(* Logix 5000 project; controller TEC_81 vendor 1 type 14 code 148 rev 36.11; software revision 36.00; part 4 of 5 *)
(* tags used below, declared in another part *)
   AbrirInterlock_conveyor_Safety : BOOL;   // Mapped green button for interlock 2 opening
   AbrirInterlock_Principal_Safety : BOOL;   // Mapped green button for interlock 1 opening
   EStops_OK : BOOL;   // E-Stop Close Loop Indicator
   Interlocks_Ok : BOOL;   // Interlocks Close Loop Indicator
   LigthCurtain_ok : BOOL;   // Light Curtains Close Loop Indicator
   MC_1_EStop : DCI_STOP;   // Status of E-Stop 1
   MC_1_EStop_Status : BOOL;   // General status of inputs
   MC_1_Interlock : DCI_STOP;   // Status of Interlock 1
   MC_1_Interlock_Status : BOOL;   // General status of inputs
   MC_1_LigthCurtain : DCI_STOP;   // Status of Light Curtain 1
   MC_1_LigthCurtain_Status : BOOL;   // General status of inputs
   MC_2_EStop : DCI_STOP;   // Status of E-Stop 2
   MC_2_EStop_Status : BOOL;   // General status of inputs
   MC_2_Interlock : DCI_STOP;   // Status of Interlock 2
   MC_2_Interlock_Status : BOOL;   // General status of inputs
   MC_2_LightCurtain_Status : BOOL;   // General status of inputs
   MC_2_LigthCurtain : DCI_STOP;   // Status of Light Curtain 2
   MC_3_EStop : DCI_STOP;   // Status of E-Stop 3
   MC_3_EStop_Status : BOOL;   // General status of inputs
   MC_4_EStop : DCI_STOP;   // Status of E-Stop 4
   MC_4_EStop_Status : BOOL;   // General status of inputs
   MC_5_EStop : DCI_STOP;   // Status of E-Stop 5
   MC_5_EStop_Status : BOOL;   // General status of inputs
   ok : BOOL;
   Ons : INT;
   Operation_Mode : BOOL;   // Operation Mode for HMI (1) Manual (0) Automatico
   Paro_Emergencia_Almacen_1 : BOOL;   // Stopping signal of Torc Off Almacen 1
   Paro_Emergencia_Almacen_2 : BOOL;   // Stopping signal of Torc Off Almacen 2
   Reset_Almacen_1_Sfty : BOOL;
   Reset_Almacen_2_Sfty : BOOL;
   Reset_Principal_Sfty : BOOL;
   Reset_Salida_1_Sfty : BOOL;
   Safety_FromTEC81 : Safety;
   SafetyReset_almacen_1 : BOOL;   // Reset status Almacen 1
   SafetyReset_almacen_2 : BOOL;   // Reset status Almacen 2
   SafetyReset_Principal : BOOL;   // Reset status salida principal
   SafetyReset_Salida_1 : BOOL;   // Reset status Salida 1
   Storage_2 : BOOL;
   Storage_3 : BOOL;
   Storage_4 : BOOL;
   Storage_5 : BOOL;
   test_com : BOOL;   // bit e comunicacion
   TEst_Leaa_Sfty : DINT;
   TOF_STO_KinetixStorage2 : TIMER;
   TT : BOOL;

PROGRAM SafetyProgram   (* main routine MainRoutine, safety *)
VAR
   dummy : BOOL;
   Lasers_OK : BOOL;   // Laser Scanner Close Loop Indicator
   LS_1 : DCI_STOP := (InputStatus := 1, RestartType := 1, ColdStartType := 1, SafetyFunction := 1, DiscrepancyTime := 200);   // Status of Laser Scanner 1
   LS_1_Status : BOOL := 1;   // General status of inputs
   LS_2 : DCI_STOP := (ChannelA := 1, ChannelB := 1, InputStatus := 1, RestartType := 1, ColdStartType := 1, SafetyFunction := 1, DiscrepancyTime := 200, O1 := 1);   // Status of Laser Scanner 2
   LS_2_Status : BOOL := 1;   // General status of inputs
   Mat_1 : DCI_STOP := (InputStatus := 1, RestartType := 1, ColdStartType := 1, SafetyFunction := 4, DiscrepancyTime := 200);   // Status of Safety Mat 1
   Mat_1_Status : BOOL := 1;   // General status of inputs
   ONS_Laser_1 : BOOL;   // One time execution for reset
   ONS_Laser_2 : BOOL;   // One time execution for reset
   ONS_Mat_1 : BOOL;   // One time execution for reset
   Output_Enable_Laser_1 : BOOL;   // General status of Laser 1
   Output_Enable_Laser_2 : BOOL;   // General status of Laser 2
   Output_Enable_Mat_1 : BOOL;   // General status of Mat 1
   Safety_Close_Loop_ok : BOOL := 1;   // General Safety Indicator
   Safety_Latch_Timer : TIMER := (PRE := 500);
   Safety_Mat_ok : BOOL;   // Safety Mat Close Loop Indicator
   Safety_Reset_General : BOOL;   // Unified General Reset
   test_1 : BOOL;
   test_21 : BOOL;
   TOF_STO_KinetixStorage1 : TIMER := (PRE := 10000, EN := 1, DN := 1);
END_VAR

ROUTINE Almacenes   (* ladder *)
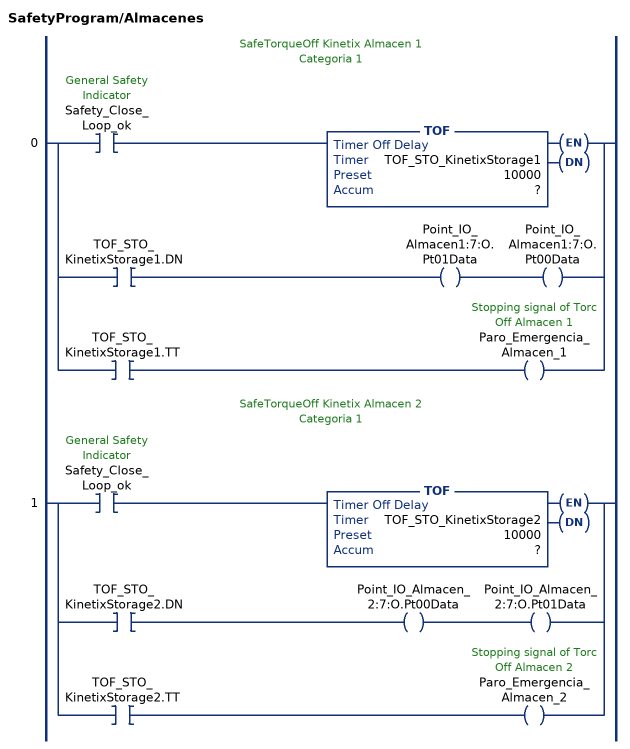
   // SafeTorqueOff Kinetix Almacen 1
   // Categoria 1
   0: [XIC(Safety_Close_Loop_ok) TOF(TOF_STO_KinetixStorage1,?,?) ,XIC(TOF_STO_KinetixStorage1.DN) OTE(Point_IO_Almacen1:7:O.Pt01Data) OTE(Point_IO_Almacen1:7:O.Pt00Data) ,XIC(TOF_STO_KinetixStorage1.TT) OTE(Paro_Emergencia_Almacen_1) ];
   // SafeTorqueOff Kinetix Almacen 2
   // Categoria 1
   1: [XIC(Safety_Close_Loop_ok) TOF(TOF_STO_KinetixStorage2,?,?) ,XIC(TOF_STO_KinetixStorage2.DN) OTE(Point_IO_Almacen_2:7:O.Pt00Data) OTE(Point_IO_Almacen_2:7:O.Pt01Data) ,XIC(TOF_STO_KinetixStorage2.TT) OTE(Paro_Emergencia_Almacen_2) ];
END_ROUTINE

ROUTINE Conveyors   (* ladder *)
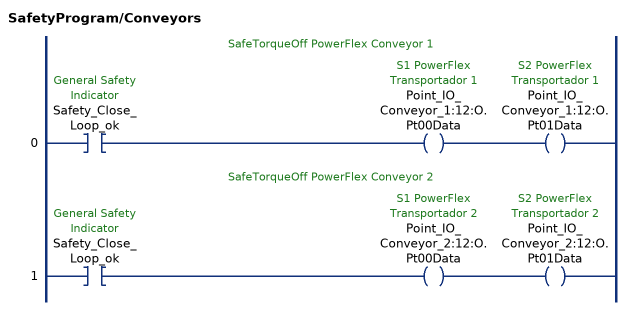
   // SafeTorqueOff PowerFlex Conveyor 1
   0: XIC(Safety_Close_Loop_ok)OTE(Point_IO_Conveyor_1:12:O.Pt00Data)OTE(Point_IO_Conveyor_1:12:O.Pt01Data);
   // SafeTorqueOff PowerFlex Conveyor 2
   1: XIC(Safety_Close_Loop_ok)OTE(Point_IO_Conveyor_2:12:O.Pt00Data)OTE(Point_IO_Conveyor_2:12:O.Pt01Data);
END_ROUTINE

ROUTINE Estops   (* ladder *)
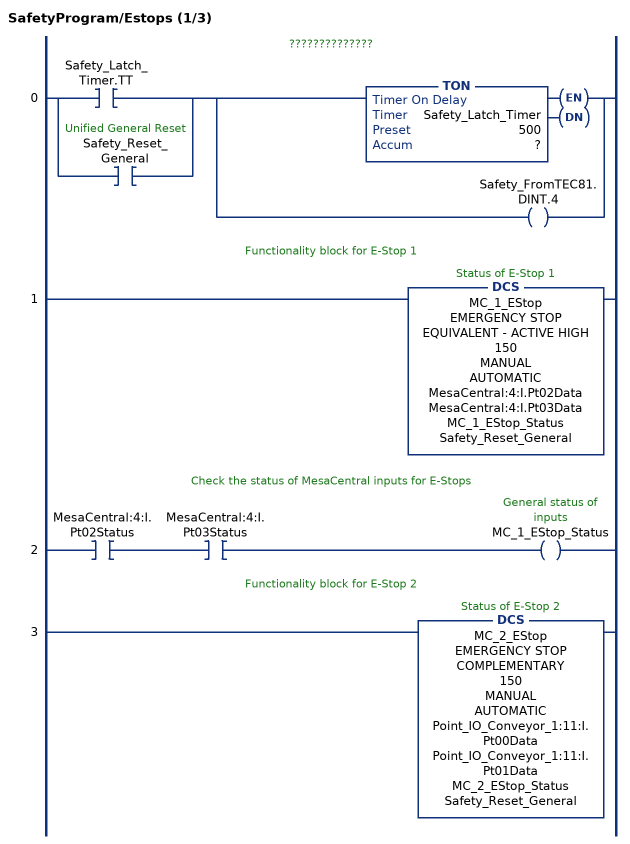
   // ??????????????
   0: [XIC(Safety_Latch_Timer.TT) ,XIC(Safety_Reset_General) ][TON(Safety_Latch_Timer,?,?) ,OTE(Safety_FromTEC81.DINT.4) ];
   // Functionality block for E-Stop 1
   1: DCS(MC_1_EStop,EMERGENCY STOP,EQUIVALENT - ACTIVE HIGH,150,MANUAL,AUTOMATIC,MesaCentral:4:I.Pt02Data,MesaCentral:4:I.Pt03Data,MC_1_EStop_Status,Safety_Reset_General);
   // Check the status of MesaCentral inputs for E-Stops
   2: XIC(MesaCentral:4:I.Pt02Status)XIC(MesaCentral:4:I.Pt03Status)OTE(MC_1_EStop_Status);
   // Functionality block for E-Stop 2
   3: DCS(MC_2_EStop,EMERGENCY STOP,COMPLEMENTARY,150,MANUAL,AUTOMATIC,Point_IO_Conveyor_1:11:I.Pt00Data,Point_IO_Conveyor_1:11:I.Pt01Data,MC_2_EStop_Status,Safety_Reset_General);
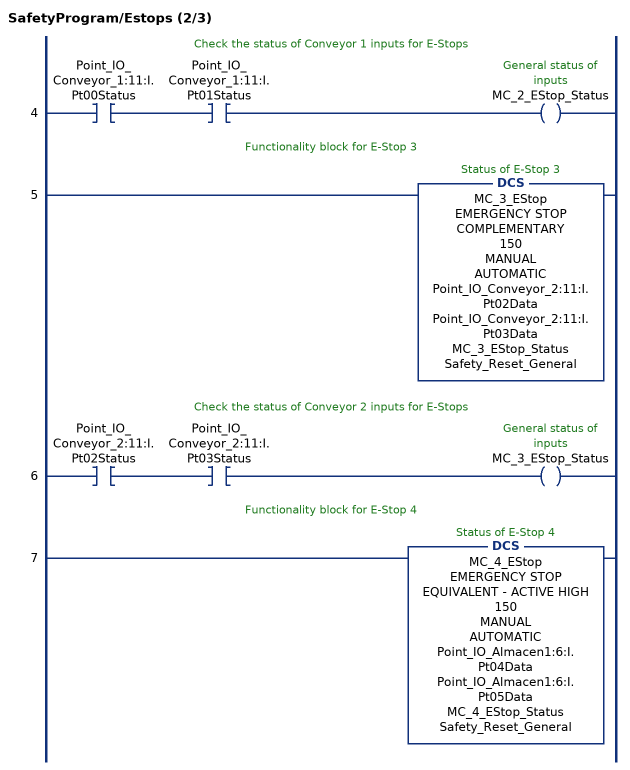
   // Check the status of Conveyor 1 inputs for E-Stops
   4: XIC(Point_IO_Conveyor_1:11:I.Pt00Status)XIC(Point_IO_Conveyor_1:11:I.Pt01Status)OTE(MC_2_EStop_Status);
   // Functionality block for E-Stop 3
   5: DCS(MC_3_EStop,EMERGENCY STOP,COMPLEMENTARY,150,MANUAL,AUTOMATIC,Point_IO_Conveyor_2:11:I.Pt02Data,Point_IO_Conveyor_2:11:I.Pt03Data,MC_3_EStop_Status,Safety_Reset_General);
   // Check the status of Conveyor 2 inputs for E-Stops
   6: XIC(Point_IO_Conveyor_2:11:I.Pt02Status)XIC(Point_IO_Conveyor_2:11:I.Pt03Status)OTE(MC_3_EStop_Status);
   // Functionality block for E-Stop 4
   7: DCS(MC_4_EStop,EMERGENCY STOP,EQUIVALENT - ACTIVE HIGH,150,MANUAL,AUTOMATIC,Point_IO_Almacen1:6:I.Pt04Data,Point_IO_Almacen1:6:I.Pt05Data,MC_4_EStop_Status,Safety_Reset_General);
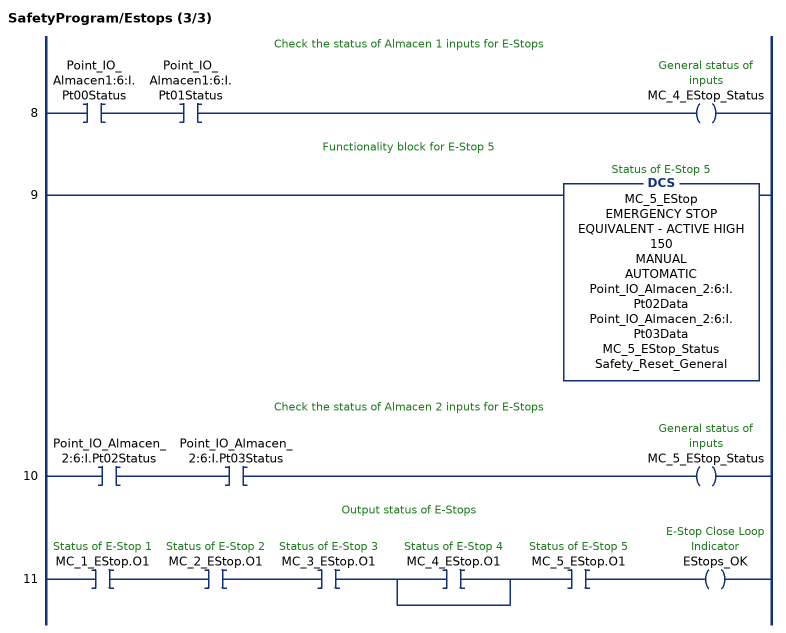
   // Check the status of Almacen 1 inputs for E-Stops
   8: XIC(Point_IO_Almacen1:6:I.Pt00Status)XIC(Point_IO_Almacen1:6:I.Pt01Status)OTE(MC_4_EStop_Status);
   // Functionality block for E-Stop 5
   9: DCS(MC_5_EStop,EMERGENCY STOP,EQUIVALENT - ACTIVE HIGH,150,MANUAL,AUTOMATIC,Point_IO_Almacen_2:6:I.Pt02Data,Point_IO_Almacen_2:6:I.Pt03Data,MC_5_EStop_Status,Safety_Reset_General);
   // Check the status of Almacen 2 inputs for E-Stops
   10: XIC(Point_IO_Almacen_2:6:I.Pt02Status)XIC(Point_IO_Almacen_2:6:I.Pt03Status)OTE(MC_5_EStop_Status);
   // Output status of E-Stops
   11: XIC(MC_1_EStop.O1)XIC(MC_2_EStop.O1)XIC(MC_3_EStop.O1)[XIC(MC_4_EStop.O1) ,]XIC(MC_5_EStop.O1)OTE(EStops_OK);
END_ROUTINE

ROUTINE External_COMM   (* ladder *)
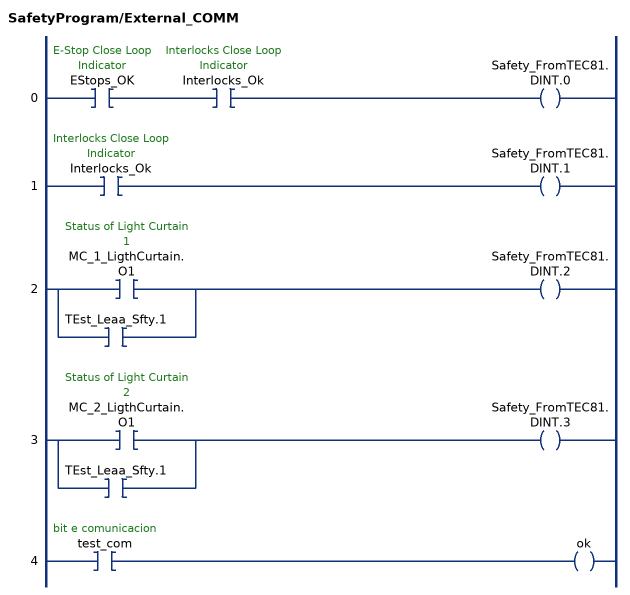
   0: XIC(EStops_OK)XIC(Interlocks_Ok)OTE(Safety_FromTEC81.DINT.0);
   1: XIC(Interlocks_Ok)OTE(Safety_FromTEC81.DINT.1);
   2: [XIC(MC_1_LigthCurtain.O1) ,XIC(TEst_Leaa_Sfty.1) ]OTE(Safety_FromTEC81.DINT.2);
   3: [XIC(MC_2_LigthCurtain.O1) ,XIC(TEst_Leaa_Sfty.1) ]OTE(Safety_FromTEC81.DINT.3);
   4: XIC(test_com)OTE(ok);
END_ROUTINE

ROUTINE Fanuc_Delta   (* ladder *)
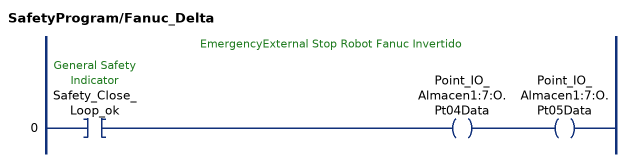
   // EmergencyExternal Stop Robot Fanuc Invertido
   0: XIC(Safety_Close_Loop_ok)OTE(Point_IO_Almacen1:7:O.Pt04Data)OTE(Point_IO_Almacen1:7:O.Pt05Data);
END_ROUTINE

ROUTINE Fanuc_Invertido   (* ladder *)
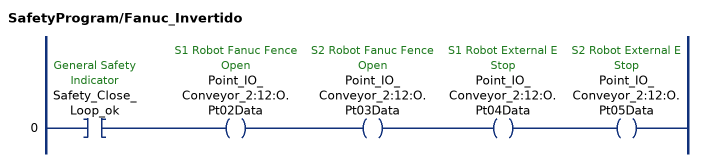
   0: XIC(Safety_Close_Loop_ok)OTE(Point_IO_Conveyor_2:12:O.Pt02Data)OTE(Point_IO_Conveyor_2:12:O.Pt03Data)OTE(Point_IO_Conveyor_2:12:O.Pt04Data)OTE(Point_IO_Conveyor_2:12:O.Pt05Data);
END_ROUTINE

ROUTINE Interlocks   (* ladder *)
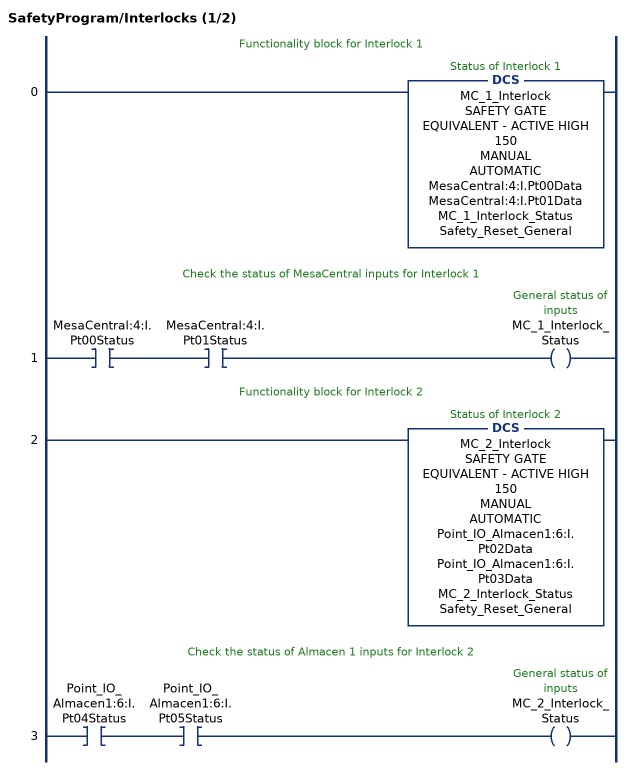
   // Functionality block for Interlock 1
   0: DCS(MC_1_Interlock,SAFETY GATE,EQUIVALENT - ACTIVE HIGH,150,MANUAL,AUTOMATIC,MesaCentral:4:I.Pt00Data,MesaCentral:4:I.Pt01Data,MC_1_Interlock_Status,Safety_Reset_General);
   // Check the status of MesaCentral inputs for Interlock 1
   1: XIC(MesaCentral:4:I.Pt00Status)XIC(MesaCentral:4:I.Pt01Status)OTE(MC_1_Interlock_Status);
   // Functionality block for Interlock 2
   2: DCS(MC_2_Interlock,SAFETY GATE,EQUIVALENT - ACTIVE HIGH,150,MANUAL,AUTOMATIC,Point_IO_Almacen1:6:I.Pt02Data,Point_IO_Almacen1:6:I.Pt03Data,MC_2_Interlock_Status,Safety_Reset_General);
   // Check the status of Almacen 1 inputs for Interlock 2
   3: XIC(Point_IO_Almacen1:6:I.Pt04Status)XIC(Point_IO_Almacen1:6:I.Pt05Status)OTE(MC_2_Interlock_Status);
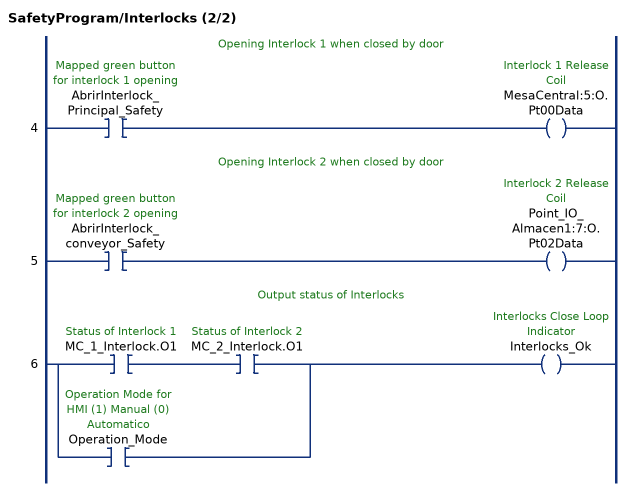
   // Opening Interlock 1 when closed by door
   4: XIC(AbrirInterlock_Principal_Safety)OTE(MesaCentral:5:O.Pt00Data);
   // Opening Interlock 2 when closed by door
   5: XIC(AbrirInterlock_conveyor_Safety)OTE(Point_IO_Almacen1:7:O.Pt02Data);
   // Output status of Interlocks
   6: [XIC(MC_1_Interlock.O1) XIC(MC_2_Interlock.O1) ,XIC(Operation_Mode) ]OTE(Interlocks_Ok);
END_ROUTINE

ROUTINE Laser_Scanner   (* ladder *)
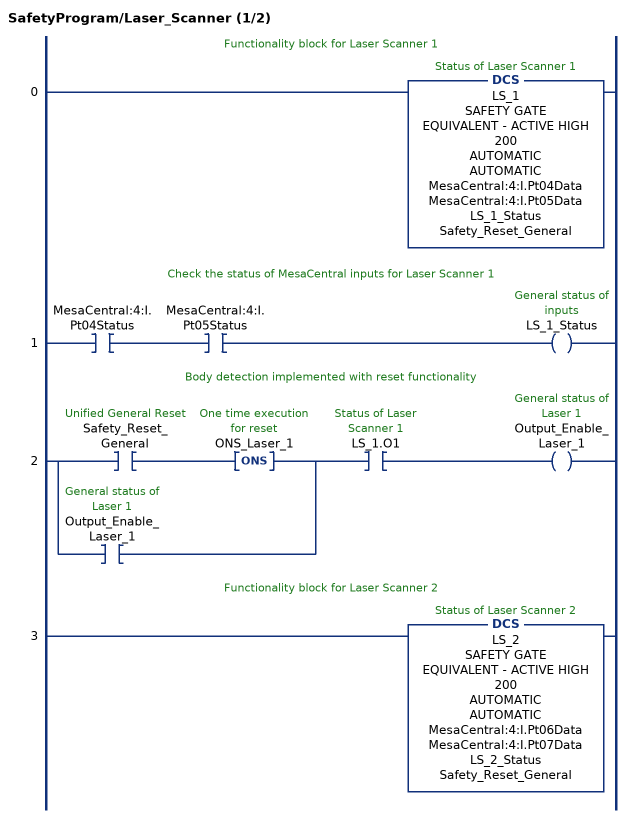
   // Functionality block for Laser Scanner 1
   0: DCS(LS_1,SAFETY GATE,EQUIVALENT - ACTIVE HIGH,200,AUTOMATIC,AUTOMATIC,MesaCentral:4:I.Pt04Data,MesaCentral:4:I.Pt05Data,LS_1_Status,Safety_Reset_General);
   // Check the status of MesaCentral inputs for Laser Scanner 1
   1: XIC(MesaCentral:4:I.Pt04Status)XIC(MesaCentral:4:I.Pt05Status)OTE(LS_1_Status);
   // Body detection implemented with reset functionality
   2: [XIC(Safety_Reset_General) ONS(ONS_Laser_1) ,XIC(Output_Enable_Laser_1) ]XIC(LS_1.O1)OTE(Output_Enable_Laser_1);
   // Functionality block for Laser Scanner 2
   3: DCS(LS_2,SAFETY GATE,EQUIVALENT - ACTIVE HIGH,200,AUTOMATIC,AUTOMATIC,MesaCentral:4:I.Pt06Data,MesaCentral:4:I.Pt07Data,LS_2_Status,Safety_Reset_General);
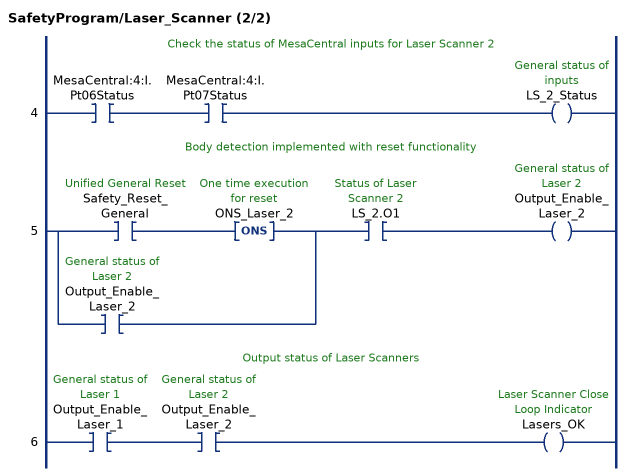
   // Check the status of MesaCentral inputs for Laser Scanner 2
   4: XIC(MesaCentral:4:I.Pt06Status)XIC(MesaCentral:4:I.Pt07Status)OTE(LS_2_Status);
   // Body detection implemented with reset functionality
   5: [XIC(Safety_Reset_General) ONS(ONS_Laser_2) ,XIC(Output_Enable_Laser_2) ]XIC(LS_2.O1)OTE(Output_Enable_Laser_2);
   // Output status of Laser Scanners
   6: XIC(Output_Enable_Laser_1)XIC(Output_Enable_Laser_2)OTE(Lasers_OK);
END_ROUTINE

ROUTINE LigthCurrtains   (* ladder *)
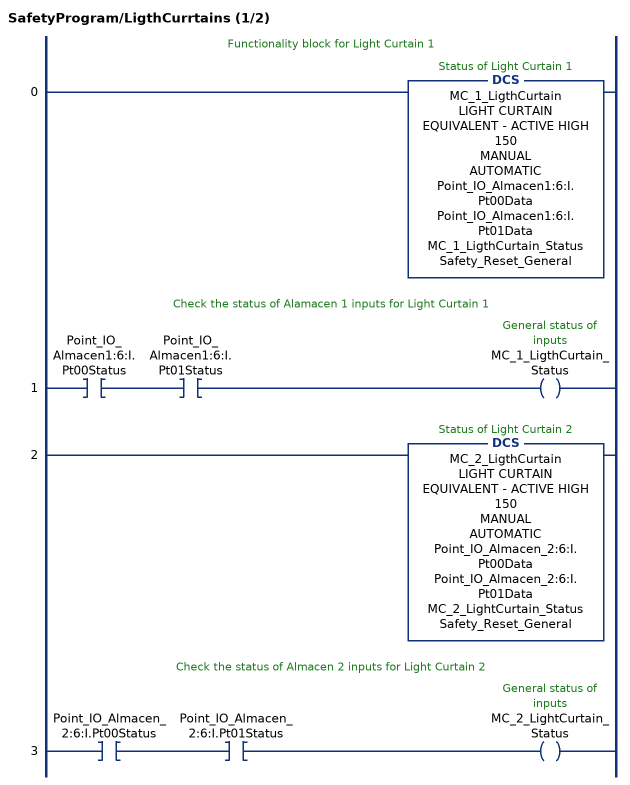
   // Functionality block for Light Curtain 1
   0: DCS(MC_1_LigthCurtain,LIGHT CURTAIN,EQUIVALENT - ACTIVE HIGH,150,MANUAL,AUTOMATIC,Point_IO_Almacen1:6:I.Pt00Data,Point_IO_Almacen1:6:I.Pt01Data,MC_1_LigthCurtain_Status,Safety_Reset_General);
   // Check the status of Alamacen 1 inputs for Light Curtain 1
   1: XIC(Point_IO_Almacen1:6:I.Pt00Status)XIC(Point_IO_Almacen1:6:I.Pt01Status)OTE(MC_1_LigthCurtain_Status);
   2: DCS(MC_2_LigthCurtain,LIGHT CURTAIN,EQUIVALENT - ACTIVE HIGH,150,MANUAL,AUTOMATIC,Point_IO_Almacen_2:6:I.Pt00Data,Point_IO_Almacen_2:6:I.Pt01Data,MC_2_LightCurtain_Status,Safety_Reset_General);
   // Check the status of Almacen 2 inputs for Light Curtain 2
   3: XIC(Point_IO_Almacen_2:6:I.Pt00Status)XIC(Point_IO_Almacen_2:6:I.Pt01Status)OTE(MC_2_LightCurtain_Status);
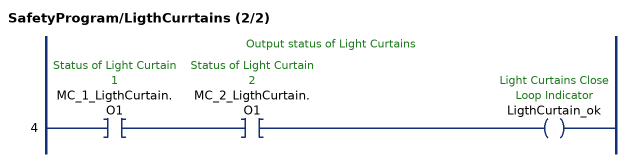
   // Output status of Light Curtains
   4: XIC(MC_1_LigthCurtain.O1)XIC(MC_2_LigthCurtain.O1)OTE(LigthCurtain_ok);
END_ROUTINE

ROUTINE MainRoutine   (* ladder *)
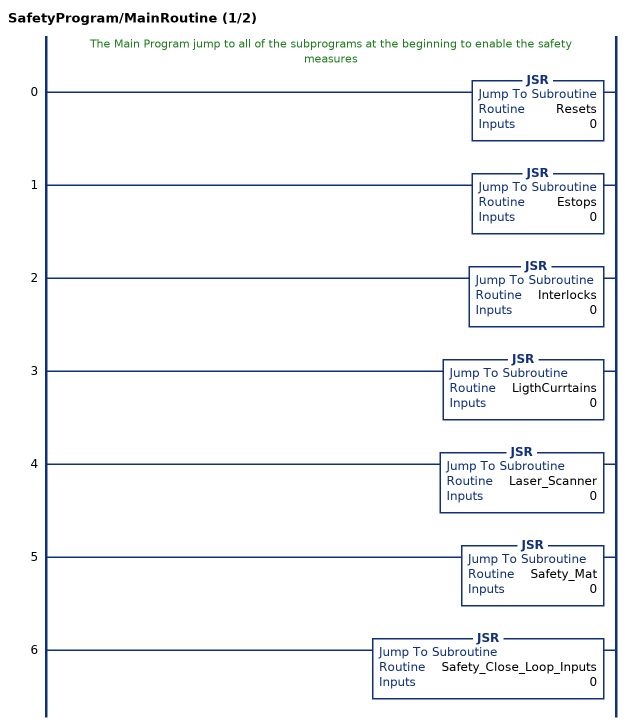
   // The Main Program jump to all of the subprograms at the beginning to enable the safety measures
   0: JSR(Resets,0);
   1: JSR(Estops,0);
   2: JSR(Interlocks,0);
   3: JSR(LigthCurrtains,0);
   4: JSR(Laser_Scanner,0);
   5: JSR(Safety_Mat,0);
   6: JSR(Safety_Close_Loop_Inputs,0);
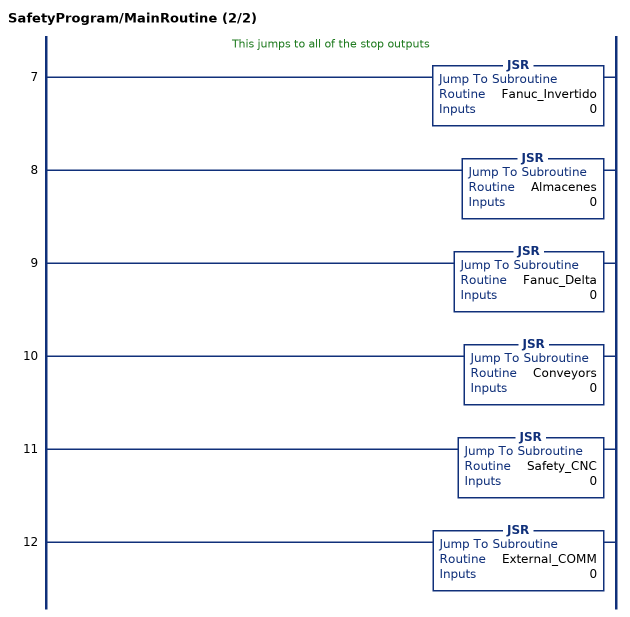
   // This jumps to all of the stop outputs
   7: JSR(Fanuc_Invertido,0);
   8: JSR(Almacenes,0);
   9: JSR(Fanuc_Delta,0);
   10: JSR(Conveyors,0);
   11: JSR(Safety_CNC,0);
   12: JSR(External_COMM,0);
END_ROUTINE

ROUTINE Resets   (* ladder *)
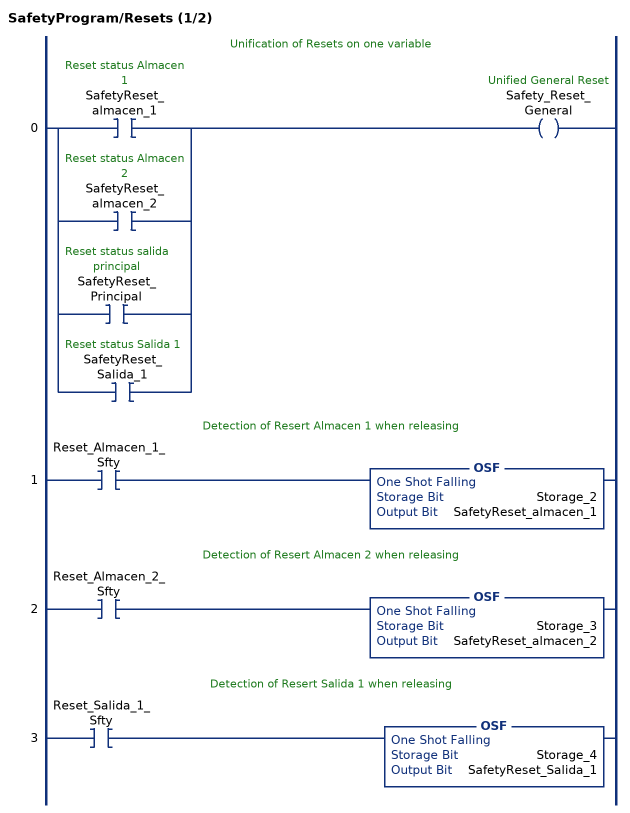
   // Unification of Resets on one variable
   0: [XIC(SafetyReset_almacen_1) ,XIC(SafetyReset_almacen_2) ,XIC(SafetyReset_Principal) ,XIC(SafetyReset_Salida_1) ]OTE(Safety_Reset_General);
   // Detection of Resert Almacen 1 when releasing
   1: XIC(Reset_Almacen_1_Sfty)OSF(Storage_2,SafetyReset_almacen_1);
   // Detection of Resert Almacen 2 when releasing
   2: XIC(Reset_Almacen_2_Sfty)OSF(Storage_3,SafetyReset_almacen_2);
   // Detection of Resert Salida 1 when releasing
   3: XIC(Reset_Salida_1_Sfty)OSF(Storage_4,SafetyReset_Salida_1);
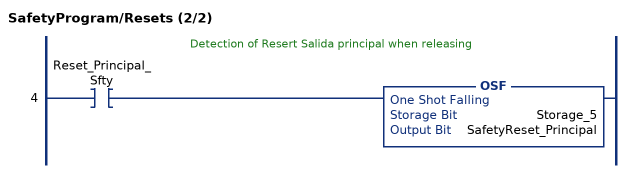
   // Detection of Resert Salida principal when releasing
   4: XIC(Reset_Principal_Sfty)OSF(Storage_5,SafetyReset_Principal);
END_ROUTINE
